INTERFACE I_JsonDataTypePack

METHOD PUBLIC RegisterWithLanguagePack
VAR_INPUT
	LanguagePack : I_JsonLanguagePack;
END_VAR
END_METHOD

END_INTERFACE

(* stored: Version 1.1.0.1, ProductVersion 3.1.4024.12
   Itf I_JsonDataTypePack: Id {c60741ea-3237-0ac6-2f76-f10f1e446198}
   Method RegisterWithLanguagePack: Id {a50b900d-258c-08bb-3c09-dc93df12a0ea} *)
